{attribute 'linkalways'} 
{attribute 'no_explicit_call' := 'This FB is a CLASS and must be accessed using methods or properties'}
{attribute 'enable_dynamic_creation'}
FUNCTION_BLOCK Node_F_VN_GetAt_ITcVnImage EXTENDS VisionNode
VAR
    ipContainer : _ITcVnContainer;
    ipElement : _ITcVnImage;
    nIndex : _ULINT(0);
    hrPrev : _HRESULT(S_OK);
    hresult : _HRESULT(S_OK);
END_VAR

METHOD PUBLIC  Clone : I_Node
VAR
	pNode : POINTER TO Node_F_VN_GetAt_ITcVnImage;
END_VAR
pNode := __NEW(Node_F_VN_GetAt_ITcVnImage);
Clone := pNode^;
END_METHOD

METHOD FB_init : BOOL
VAR_INPUT
	bInitRetains : BOOL; // if TRUE, the retain variables are initialized (warm start / cold start)
	bInCopyCode : BOOL;  // if TRUE, the instance afterwards gets moved into the copy code (online change)
END_VAR
AddInput('ipContainer', ipContainer);
AddParameter('nIndex', nIndex);
AddInput('hrPrev', hrPrev);
AddOutput('ipElement', ipElement);
AddOutput('hresult',hresult);
END_METHOD

METHOD PROTECTED OnExecute
hresult.Value := F_VN_GetAt_ITcVnImage(
    ipContainer := ipContainer.Value,
    ipElement := ipElement.Value,
    nIndex := nIndex.Value,
    hrPrev:= hrPrev.Value);
END_METHOD

METHOD PUBLIC PreExecutionCheck
VAR_INPUT
	Check : I_PreExecutionChecks;
END_VAR
Check.IsTrue(ipContainer.IsValid, 'ipContainer must be a valid container');
Check.IsTrue(ipContainer.IsType(TC_GLOBAL_CONST_LIST.ContainerType_Vector_ITcVnImage), 'ipContainer contains incorrect type');
END_METHOD

END_FUNCTION_BLOCK

(* stored: Version 1.1.0.1, ProductVersion 3.1.4026.13
   POU Node_F_VN_GetAt_ITcVnImage: Id {b8b8d385-5631-4647-b0c5-53853d2296c4}, SpecialFunc None
   Folder Constructor: Id {f1830bea-6e7b-4aad-826f-73bc786745db}
   Method Clone: Id {20530fbe-2c91-45e2-ba6c-d7015487b9d8}
   Method FB_init: Id {513a3a65-f49c-4315-b0ef-a3fd40d23710}
   Method OnExecute: Id {68436676-d0ea-4c9e-ad73-a0ae4e41da14}
   Method PreExecutionCheck: Id {566e94dc-e871-43d2-8b3e-4c7b7ac0ae4a} *)
